// TIA Portal V19 export
TYPE "LEXCHANGETRAY_typeNgConveyorEm_toHandlingXyzRecieve"
// stored: Access Published
   STRUCT
      feedback { S7_SetPoint := 'True'} : "LEXCHANGETRAY_typeHandlingXyzEm_toNgConveyorFeedback";
      req { S7_SetPoint := 'True'} : "LEXCHANGETRAY_typeHandlingXyzEm_toNgConveyoReq";
   END_STRUCT;
END_TYPE
